INTERFACE IDevice EXTENDS Core.IObject, ISimulatable

METHOD EmergncyStop
END_METHOD

METHOD HandleFault
END_METHOD

METHOD Initialize : BOOL
END_METHOD

{attribute 'monitoring' := 'call'}
{attribute 'OPC.UA.DA' := '1'}
{attribute 'OPC.UA.DA.Access' := '1'}
PROPERTY FINAL LocalSimulationMode : BOOL
GET
END_GET
END_PROPERTY

END_INTERFACE

(* stored: Version 1.1.0.1
   Itf IDevice: Id {f88c7d43-a687-48ea-a56a-1df42b081949}
   Method EmergncyStop: Id {09eae555-d338-43f3-9cee-0c8fc29c0a1d}
   Method HandleFault: Id {48c1b4f0-66ed-4281-8ac8-d4a7eb0f6d97}
   Method Initialize: Id {fe44ff0a-9dac-4461-a04f-f97c80ce5b13}
   Property LocalSimulationMode: Id {9cb3fd13-88f3-4dac-8e8e-97bd1d1858a7}
   Get Get: Id {eb142456-4e4f-478d-8119-ee9bf42d69ac} *)
